FUNCTION_BLOCK FB_PressureSensor EXTENDS FB_Sensor
VAR_INPUT
END_VAR
VAR_OUTPUT
	fPressure : REAL; //measured pressure in bar
END_VAR
VAR	
	//I/O-Links
	nPressure_IN AT %I* : INT;
END_VAR

METHOD GetState_AI : BOOL
VAR_INPUT
END_VAR
VAR
END_VAR
// scaling to [0,6000]
fPressure := (INT_TO_REAL(nPressure_IN))*0.1831/1000 ;

//sensor state
sensorState.fValue := fPressure;
sensorState.sUnit := 'bar';
END_METHOD

END_FUNCTION_BLOCK

(* stored: Version 1.1.0.1, ProductVersion 3.1.4024.10
   POU FB_PressureSensor: Id {7044f823-1ed9-4edf-a9f3-50efcf49ac23}, SpecialFunc None
   Method GetState_AI: Id {2f26965c-ca17-4f24-ac3f-b491df8f99e3} *)
